FUNCTION MMIN_TO_MMS : LREAL
VAR_INPUT
	IN														:	LREAL;
END_VAR
VAR
END_VAR

IF IN = 0.0
THEN
	MMIN_TO_MMS 											:= 0.0;
ELSE            											
	MMIN_TO_MMS 											:= IN * 1000.0 / 60.0	;
END_IF

END_FUNCTION

(* stored: Version 1.1.0.1, ProductVersion 3.1.4024.12
   POU MMIN_TO_MMS: Id {30384bd9-2575-45ce-b3ea-e53b9dcfa6ae}, SpecialFunc None *)
